// Mitsubishi GX Works2 project: z13   PLC: Q02/Q02H

PROGRAM MAIN
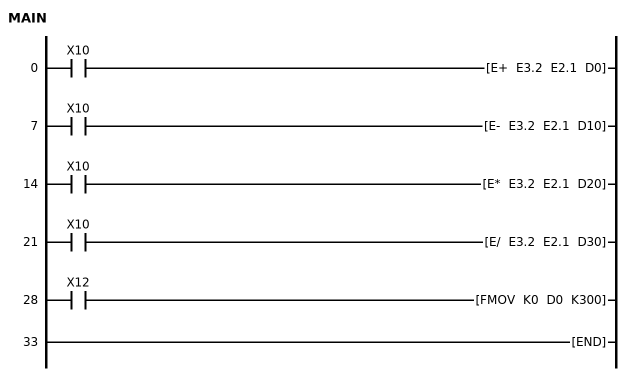
0     LD      X10
      E+      E3.2 E2.1 D0
7     LD      X10
      E-      E3.2 E2.1 D10
14    LD      X10
      E*      E3.2 E2.1 D20
21    LD      X10
      E/      E3.2 E2.1 D30
28    LD      X12
      FMOV    K0 D0 K300
33    END
END_PROGRAM
